(* PLC project Generator Governor and Program, Blank VGP 1.0 *)
(* stored: creationDateTime 2016-05-18T21:14:07, modificationDateTime 2020-06-05T23:07:53 *)

FUNCTION_BLOCK ControllerFunc1
  VAR_INPUT
    omega : INT;
    gain : INT;
    Reference : INT;
    on_off : BOOL;
  END_VAR
  VAR_OUTPUT
    act_com : INT := 0;
    act_com0 : INT := 0;
  END_VAR
  VAR
    U : REAL := 0.0;
    Ga : REAL := 0.0;
    REF : REAL := 1.0;
    ERR : REAL := 0.0;
    X1 : REAL := 0.0;
    X2 : REAL := 0.0;
    Y : REAL := 0.0;
    Y2 : REAL := 0.0;
    Xtemp : REAL := 0.0;
    A11 : REAL := 0.4337;
    A12 : REAL := -36.16;
    A21 : REAL := 0.007232;
    A22 : REAL := 0.7954;
    C1 : REAL := 1000.0;
    C2 : REAL := 5000.0;
    Dd : REAL := 0.0;
    B1 : REAL := 0.007232;
    B2 : REAL := 0.00004093;
    E_k_1 : REAL := 0.0;
    E_k_2 : REAL := 0.0;
    Y_k_1 : REAL := 0.0;
    Y_k_2 : REAL := 0.0;
    tfa0 : REAL := 9.518;
    tfa1 : REAL := -8.448;
    tfb0 : REAL := 1.0;
    tfb1 : REAL := -0.2977;
    tfb2 : REAL := 0.3679;
  END_VAR

            (* Convert the input appropriately to Input *)

(* Data Dictionary
E_k_1 = e[k - 1]
E_k_2 = e[k - 2]
Y_k_1 = e[k - 1]
Y_k_2 = e[k - 2]
*)


U := INT_TO_REAL(omega); 
Ga := INT_TO_REAL(Gain);
U := U - 10000.0; 
U := U / 10000.0;

Y := REF - U;
ERR := REF - U;
Y2 := 1.0/tfb0 * (tfa0*E_k_1 + tfa1*E_k_2 - b1*Y_k_1 - b2*Y_k_2);
 
(* Prepare variables for next iteration *)
E_k_2 := E_k_1;
E_k_1 := ERR;
Y_k_2 := Y_k_1;
Y_k_1 := Y2;



(* Now the Algorithm Performs an Iteration*)
(* Y := C1*X1 + C2*X2 + Dd*ERR; *)
(* Xtemp := X1; *)
(* X1 := A11*X1 + A12*X2 + B1*ERR; *)
(* X2 := A21*Xtemp + A22*X2 + B2*ERR; *)

Y := Y * Ga;
Y := Y * 10000.0;
Y := Y + 10000.0;

Y2 := Y2 * Ga;
Y2 := Y2 * 10000.0;
Y2 := Y2 + 10000.0; 

act_com := REAL_TO_INT(Y);
act_com0 := REAL_TO_INT(Y2);

(* act_com := omega; *)
          
END_FUNCTION_BLOCK

FUNCTION_BLOCK ControllerFunc
  VAR_INPUT
    omega : UINT;
    gain : UINT;
    Reference : UINT := 10000;
  END_VAR
  VAR
    act_com : UINT := 0;
  END_VAR
  VAR_OUTPUT
    act_com0 : UINT := 0;
  END_VAR
  VAR
    U : REAL := 0.0;
    Ga : REAL := 0.0;
    REF : REAL := 1.0;
    ERR : REAL := 0.0;
    X1 : REAL := 0.0;
    X2 : REAL := 0.0;
    Y : REAL := 0.0;
    Y2 : REAL := 0.0;
    Xtemp : REAL := 0.0;
    A11 : REAL := 0.4337;
    A12 : REAL := -36.16;
    A21 : REAL := 0.007232;
    A22 : REAL := 0.7954;
    C1 : REAL := 1000.0;
    C2 : REAL := 5000.0;
    Dd : REAL := 0.0;
    B1 : REAL := 0.007232;
    B2 : REAL := 0.00004093;
    E_k_1 : REAL := 0.0;
    E_k_2 : REAL := 0.0;
    Y_k_1 : REAL := 0.0;
    Y_k_2 : REAL := 0.0;
    tfa0 : REAL := 9.518;
    tfa1 : REAL := -8.448;
    tfb0 : REAL := 1.0;
    tfb1 : REAL := -0.2977;
    tfb2 : REAL := 0.3679;
  END_VAR

            (* Convert the input appropriately to Input *)

(* Data Dictionary
E_k_1 = e[k - 1]
E_k_2 = e[k - 2]
Y_k_1 = e[k - 1]
Y_k_2 = e[k - 2]
*)


U := UINT_TO_REAL(omega); 
Ga := UINT_TO_REAL(Gain);
REF := UINT_TO_REAL(Reference);
REF := REF / 10000.0;
U := U - 10000.0; 
U := U / 1000.0;

Y := REF - U;
ERR := REF - U;
(* ERR := 0.50 - U;*)
Y2 := 1.0/tfb0 * (tfa0*E_k_1 + tfa1*E_k_2 - tfb1*Y_k_1 - tfb2*Y_k_2);
 
(* Prepare variables for next iteration *)
E_k_2 := E_k_1;
E_k_1 := ERR;
Y_k_2 := Y_k_1;
Y_k_1 := Y2;



(* Now the Algorithm Performs an Iteration*)
(* Y := C1*X1 + C2*X2 + Dd*ERR; *)
(* Xtemp := X1; *)
(* X1 := A11*X1 + A12*X2 + B1*ERR; *)
(* X2 := A21*Xtemp + A22*X2 + B2*ERR; *)

Y := Y * Ga;
Y := Y * 1000.0;
Y := Y + 10000.0;

Y2 := Y2 * Ga;
Y2 := Y2 * 1000.0;
Y2 := Y2 + 10000.0; 

If Y2 > 65000.0 THEN
  Y2 := 65000.0;
END_IF;
  
IF Y2 < 0.0 THEN
    Y2 := 0.0;
END_IF;
(* act_com := REAL_TO_INT(Y); *)
act_com0 := REAL_TO_UINT(Y2);

(* act_com := omega; *)
          
END_FUNCTION_BLOCK

PROGRAM My_Program
  VAR
    act_com AT %QW0 : UINT;
    act_com0 AT %QW1 : UINT;
    Gain AT %QW2 : UINT := 40;
    vrms0 AT %QW3 : UINT := 0;
    Reference AT %QW4 : UINT := 10000;
    vrms_max AT %QW5 : UINT := 20000;
    irms_max AT %QW6 : UINT := 20000;
    Oil_min AT %QW7 : UINT := 10;
    Temp_min AT %QW8 : UINT := 0;
    Temp_max AT %QW9 : UINT := 500;
    rpm_max AT %QW10 : UINT := 20000;
    vrms AT %IW0 : UINT;
    Irms AT %IW1 : UINT;
    Frequency AT %IW2 : UINT;
    RPM AT %IW3 : UINT;
    Fuel AT %IW4 : UINT;
    Oil AT %IW5 : UINT := 10;
    Temp AT %IW6 : UINT;
    omega AT %IW7 : UINT := 0;
    switch AT %QX0.0 : BOOL := 0;
    onoff AT %QX0.1 : BOOL := 0;
    Override AT %QX0.2 : BOOL := 0;
    Fault AT %QX0.3 : BOOL := 0;
    Reset AT %QX0.4 : BOOL := 0;
    Fault2 AT %QX0.5 : BOOL := 0;
  END_VAR
  VAR
    ControllerFunc0 : ControllerFunc;
  END_VAR

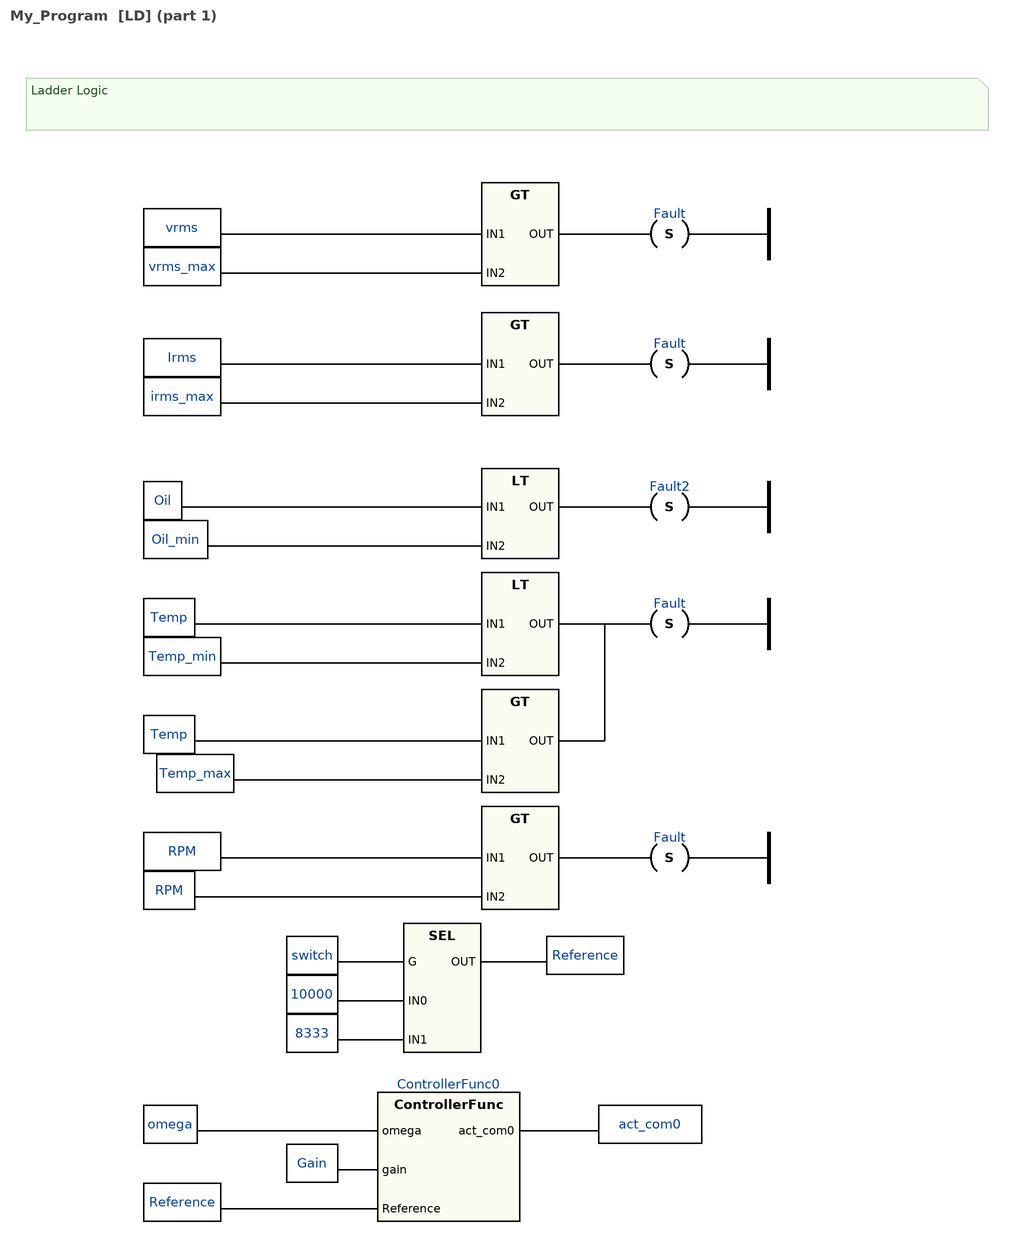
(* LD diagram, written out as Structured Text *)
(* Ladder Logic *)
IF vrms > vrms_max THEN Fault := TRUE; END_IF;
IF Irms > irms_max THEN Fault := TRUE; END_IF;
IF Oil < Oil_min THEN Fault2 := TRUE; END_IF;
IF Temp < Temp_min OR Temp > Temp_max THEN Fault := TRUE; END_IF;
IF RPM > RPM THEN Fault := TRUE; END_IF;
Reference := SEL(switch, 10000, 8333);
ControllerFunc0(omega := omega, gain := Gain, Reference := Reference);
act_com0 := ControllerFunc0.act_com0;
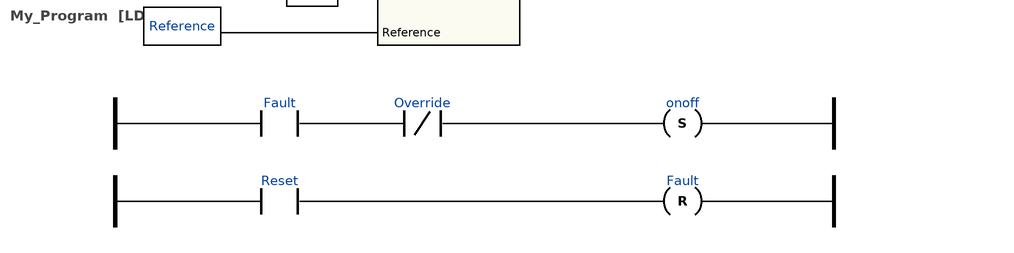
IF Fault AND NOT Override THEN onoff := TRUE; END_IF;
IF Reset THEN Fault := FALSE; END_IF;
END_PROGRAM

FUNCTION_BLOCK Controller
  VAR_INPUT
    omega : INT;
    gain : INT;
  END_VAR
  VAR_OUTPUT
    act_com : INT;
  END_VAR
  VAR
    U : REAL := 0.0;
    Ga : REAL := 0.0;
    REF : REAL := 1.0;
    ERR : REAL := 0.0;
    Y : REAL := 0.0;
    X1 : REAL := 0.0;
    X2 : REAL := 0.0;
    Xtemp : REAL := 0.0;
    A11 : REAL := 0.4337;
    A12 : REAL := -36.16;
    A21 : REAL := 0.007232;
    A22 : REAL := 0.7954;
    C1 : REAL := 1000.0;
    C2 : REAL := 5000.0;
    Dd : REAL := 0.0;
    B1 : REAL := 0.007232;
    B2 : REAL := 0.00004093;
  END_VAR

            (* Convert the input appropriately to Input *)
U := INT_TO_REAL(omega); 
Ga := INT_TO_REAL(Gain);
U := U - 1000.0; 
U := U / 1000.0;

(* ERR := REF - U; *)
ERR := 0.8333 - U;


(* Now the Algorithm Performs an Iteration*)
Y := C1*X1 + C2*X2 + Dd*ERR;
Xtemp := X1;
X1 := A11*X1 + A12*X2 + B1*ERR;
X2 := A21*Xtemp + A22*X2 + B2*ERR;
Y := Y * Ga;

Y := Y * 1000.0;
Y := Y + 10000.0; 
act_com := REAL_TO_INT(Y);

(* act_com := omega; *)
          
END_FUNCTION_BLOCK

CONFIGURATION Config0
  RESOURCE Res0 ON PLC
    TASK TaskMain(INTERVAL := T#200ms, PRIORITY := 0);
    PROGRAM Inst0 WITH TaskMain : My_Program;
  END_RESOURCE
END_CONFIGURATION
